FUNCTION_BLOCK ADSDataService IMPLEMENTS ITF_MachineDataService
VAR
	_messageSent : int;
END_VAR

METHOD SendStatus : INT
VAR_INPUT
	Status : INT;
END_VAR
_messageSent := Status;
END_METHOD

END_FUNCTION_BLOCK

(* stored: Version 1.1.0.1, ProductVersion 3.1.4024.12
   POU ADSDataService: Id {b7572e9b-04d7-4be9-9c2f-3e8319bd29b7}, SpecialFunc None
   Method SendStatus: Id {899a0856-473c-40e4-9573-a1d93df990d4} *)
